FUNCTION_BLOCK FBRealtimeSupport
///SDOC/////////////////////////////////////////////////////////////////////////
//
//  FBRealtimeSupport.TcPOU      - Function Block - Real-time diagnostic data with analog data - AVT PLC 
//						Version 1
//  Author:         Mark Colvin                         Date: Sept 5, 2018
//
//	Beckhoff TC3 Structured Text for CX8190 PLC
//
//	includes features:
//		10 inker enables
///////////////////////////////////////////////////////////////////////SDOCEND//
VAR_INPUT
END_VAR
VAR_OUTPUT
END_VAR
VAR
	// === LOCAL DATA === NOT saved over power cycles
	Index		:WORD;	//temp fountain index 
	wCycleCount	:WORD;	//cycle count for ON time for inker/water adjustments
	nActualScaled: INT;
	iActual: INT;
	w_output_incr	:INT;
END_VAR
VAR CONSTANT
	FTN1		:WORD:= 0;	//constants for fountain indexes fro IO arrays in TBs
	FTN2		:WORD:= 1;
	FTN3		:WORD:= 2;
	FTN4		:WORD:= 3;
	FTN5		:WORD:= 4;
	FTN6		:WORD:= 5;
	FTN7		:WORD:= 6;
	FTN8		:WORD:= 7;
	FTN9		:WORD:= 8;
	FTN10	:WORD:= 9;
	wMotorTimeOn :WORD:=500;  //wMotorTimeOn, how long the output is ON for ONE motor adjustment(+ or -), 1000 = 1second
END_VAR


	 CASE GVL.mb_Output_Registers[GVL.REALTIME_DATA_SELECTION] OF		//this is user selection of fountain control to inspect/modify
	 0:	//do nothing here
	 
	 // Inker analog inputs and outputs
	 1:	Index := FTN1;		//assign temp index
		CASE GVL.mb_Output_Registers[GVL.INKERHARDWARETYPE] OF
(* 		GVL.SWPWTR_TIME:
			//GVL.mb_Output_Registers[GVL.REALTIME_PLC_A2D] :=	0;	//nothing to read with FB circuit, just move motor
			IF GVL.mb_Output_Coils[GVL.REALTIME_ADVANCE] THEN		//move the motor forward
				IF TRUE THEN							//test the FB for limit - can't do this, pass through
					GVL.mb_Output_Coils[GVL.InkSweepRUN +(FTN1 * GVL.BOOLRUNTIMEGROUPSIZE)] := 	TRUE; //next RUN will force to console target
					GVL_IO.InkMotorFwd[FTN1] := TRUE;				// turn on the advance output
					GVL_IO.InkMotorRvs[FTN1] := FALSE;
					wCycleCount := wCycleCount + 1;
					IF wCycleCount > wMotorTimeOn THEN				//done with timer?
						GVL_IO.InkMotorFwd[FTN1] := FALSE;		//turn off outputs
						GVL_IO.InkMotorRvs[FTN1] := FALSE;
						GVL.mb_Output_Coils[GVL.REALTIME_ADVANCE] := FALSE; // reset the advance boolean
						wCycleCount := 0;					//reset the timer counter						
					END_IF
				END_IF
			END_IF
			IF GVL.mb_Output_Coils[GVL.REALTIME_RETARD] THEN
				IF TRUE THEN							//test the FB for limit - can't do this, pass through
					GVL.mb_Output_Coils[GVL.InkSweepRUN +(FTN1 * GVL.BOOLRUNTIMEGROUPSIZE)] := 	TRUE; //next RUN will force to console target
					GVL_IO.InkMotorFwd[FTN1] := FALSE;				// turn on the reverse output
					GVL_IO.InkMotorRvs[FTN1] := TRUE;
					wCycleCount := wCycleCount + 1;
					IF wCycleCount > wMotorTimeOn THEN				//done with timer?
						GVL_IO.InkMotorFwd[FTN1] := FALSE;		//turn off outputs
						GVL_IO.InkMotorRvs[FTN1] := FALSE;
						GVL.mb_Output_Coils[GVL.REALTIME_RETARD] := FALSE; // reset the reverse boolean
						wCycleCount := 0;					//reset the timer counter						
					END_IF
				END_IF
			END_IF
		GVL.SWPWTR_FB:
			GVL.mb_Output_Registers[GVL.REALTIME_PLC_A2D] :=	INT_TO_WORD(GVL_IO.InkInput[FTN1]);
			IF GVL.mb_Output_Coils[GVL.REALTIME_ADVANCE] THEN		//move the motor forward
				IF INT_TO_WORD(GVL_IO.InkInput[FTN1]) < 32000 THEN				//test the FB for limit - assumes 32767 is max of 10 VDC
					GVL.mb_Output_Coils[GVL.InkSweepRUN +(FTN1 * GVL.BOOLRUNTIMEGROUPSIZE)] := 	TRUE; //next RUN will force to console target
					GVL_IO.InkMotorFwd[FTN1] := TRUE;				// turn on the advance output
					GVL_IO.InkMotorRvs[FTN1] := FALSE;
					wCycleCount := wCycleCount + 1;
					IF wCycleCount > wMotorTimeOn THEN				//done with timer?
						GVL_IO.InkMotorFwd[FTN1] := FALSE;		//turn off outputs
						GVL_IO.InkMotorRvs[FTN1] := FALSE;
						GVL.mb_Output_Coils[GVL.REALTIME_ADVANCE] := FALSE; // reset the advance boolean
						wCycleCount := 0;					//reset the timer counter	
						//  curr % sweep   curr ticks - min tick allowed      max sweep %            max ticks allowed      min ticks allowed
						GVL.mb_Output_Registers[GVL.SWEEPTRIMONPRESS + (FTN10 * GVL.WORDRUNTIMEGROUPSIZE)]	:= (INT_TO_WORD(GVL_IO.InkInput[FTN1]) - GVL.w_InkInputIntMin[FTN10]) * 
								(GVL.mb_Output_Registers[GVL.MAXSWEEPTRIM]+1) / (GVL.w_InkInputIntMax[FTN10] - GVL.w_InkInputIntMin[FTN10]);
						//need the onpress setting pointed to the current % sweep of the positioner
					END_IF
				END_IF
			END_IF
			IF GVL.mb_Output_Coils[GVL.REALTIME_RETARD] THEN
				IF INT_TO_WORD(GVL_IO.InkInput[FTN1]) > 800 THEN				//test the FB for limit - assumes 32767 is max of 10 VDC
					GVL.mb_Output_Coils[GVL.InkSweepRUN +(FTN1 * GVL.BOOLRUNTIMEGROUPSIZE)] := 	TRUE; //next RUN will force to console target
					GVL_IO.InkMotorFwd[FTN1] := FALSE;				// turn on the reverse output
					GVL_IO.InkMotorRvs[FTN1] := TRUE;
					wCycleCount := wCycleCount + 1;
					IF wCycleCount > wMotorTimeOn THEN				//done with timer?
						GVL_IO.InkMotorFwd[FTN1] := FALSE;		//turn off outputs
						GVL_IO.InkMotorRvs[FTN1] := FALSE;
						GVL.mb_Output_Coils[GVL.REALTIME_RETARD] := FALSE; // reset the reverse boolean
						wCycleCount := 0;					//reset the timer counter						
						//  curr % sweep   curr ticks - min tick allowed      max sweep %            max ticks allowed      min ticks allowed
						GVL.mb_Output_Registers[GVL.SWEEPTRIMONPRESS + (FTN1 * GVL.WORDRUNTIMEGROUPSIZE)]	:= (INT_TO_WORD(GVL_IO.InkInput[FTN1]) - GVL.w_InkInputIntMin[FTN1]) * 
								(GVL.mb_Output_Registers[GVL.MAXSWEEPTRIM]+1) / (GVL.w_InkInputIntMax[FTN1] - GVL.w_InkInputIntMin[FTN1]);
						//need the onpress setting pointed to the current % sweep of the positioner
					END_IF
				END_IF
			END_IF
		GVL.SWPWTR_OUTPUT:
			GVL.mb_Output_Registers[GVL.REALTIME_PLC_A2D] :=	INT_TO_WORD(GVL_IO.InkSweepOut[FTN1]);
			IF( GVL.b_DINTInput) THEN									//how big should the adv / ret control increment be?
				w_output_incr :=  DINT_TO_INT(GVL.d_DINT10V / 100);
			ELSE
				w_output_incr := (GVL.i_INT10V / 100);
			END_IF
			IF GVL.mb_Output_Coils[GVL.REALTIME_ADVANCE] THEN
				IF (GVL_IO.InkSweepOut[FTN1]) < (w_output_incr *100) THEN
					GVL.mb_Output_Coils[GVL.InkSweepRUN +(FTN1 * GVL.BOOLRUNTIMEGROUPSIZE)] := 	TRUE; //next RUN will force to console target
					GVL_IO.InkSweepOut[FTN1] := (GVL_IO.InkSweepOut[FTN1]) + w_output_incr;
				END_IF
				GVL.mb_Output_Coils[GVL.REALTIME_ADVANCE] := FALSE;
			END_IF
			IF GVL.mb_Output_Coils[GVL.REALTIME_RETARD] THEN
				IF (GVL_IO.InkSweepOut[FTN1]) > w_output_incr THEN
					GVL.mb_Output_Coils[GVL.InkSweepRUN +(FTN1 * GVL.BOOLRUNTIMEGROUPSIZE)] := 	TRUE; //next RUN will force to console target
					GVL_IO.InkSweepOut[FTN1] := (GVL_IO.InkSweepOut[FTN1]) - w_output_incr;
				END_IF
				GVL.mb_Output_Coils[GVL.REALTIME_RETARD] := FALSE;
			END_IF			
 *)
		GVL.SWPWTR_BRIDGE:

		END_CASE
	 2:	Index := FTN2;		//assign temp index
		CASE GVL.mb_Output_Registers[GVL.INKERHARDWARETYPE] OF
(* 		GVL.SWPWTR_TIME:
			//GVL.mb_Output_Registers[GVL.REALTIME_PLC_A2D] :=	0;	//nothing to read with FB circuit, just move motor
			IF GVL.mb_Output_Coils[GVL.REALTIME_ADVANCE] THEN		//move the motor forward
				IF TRUE THEN							//test the FB for limit - can't do this, pass through
					GVL.mb_Output_Coils[GVL.InkSweepRUN +(FTN2 * GVL.BOOLRUNTIMEGROUPSIZE)] := 	TRUE; //next RUN will force to console target
					GVL_IO.InkMotorFwd[FTN2] := TRUE;				// turn on the advance output
					GVL_IO.InkMotorRvs[FTN2] := FALSE;
					wCycleCount := wCycleCount + 1;
					IF wCycleCount > wMotorTimeOn THEN				//done with timer?
						GVL_IO.InkMotorFwd[FTN2] := FALSE;		//turn off outputs
						GVL_IO.InkMotorRvs[FTN2] := FALSE;
						GVL.mb_Output_Coils[GVL.REALTIME_ADVANCE] := FALSE; // reset the advance boolean
						wCycleCount := 0;					//reset the timer counter						
					END_IF
				END_IF
			END_IF
			IF GVL.mb_Output_Coils[GVL.REALTIME_RETARD] THEN
				IF TRUE THEN							//test the FB for limit - can't do this, pass through
					GVL.mb_Output_Coils[GVL.InkSweepRUN +(FTN2 * GVL.BOOLRUNTIMEGROUPSIZE)] := 	TRUE; //next RUN will force to console target
					GVL_IO.InkMotorFwd[FTN2] := FALSE;				// turn on the reverse output
					GVL_IO.InkMotorRvs[FTN2] := TRUE;
					wCycleCount := wCycleCount + 1;
					IF wCycleCount > wMotorTimeOn THEN				//done with timer?
						GVL_IO.InkMotorFwd[FTN2] := FALSE;		//turn off outputs
						GVL_IO.InkMotorRvs[FTN2] := FALSE;
						GVL.mb_Output_Coils[GVL.REALTIME_RETARD] := FALSE; // reset the reverse boolean
						wCycleCount := 0;					//reset the timer counter						
					END_IF
				END_IF
			END_IF
		GVL.SWPWTR_FB:
			GVL.mb_Output_Registers[GVL.REALTIME_PLC_A2D] :=	INT_TO_WORD(GVL_IO.InkInput[FTN2]);
			IF GVL.mb_Output_Coils[GVL.REALTIME_ADVANCE] THEN		//move the motor forward
				IF INT_TO_WORD(GVL_IO.InkInput[FTN2]) < 32000 THEN				//test the FB for limit - assumes 32767 is max of 10 VDC
					GVL.mb_Output_Coils[GVL.InkSweepRUN +(FTN2 * GVL.BOOLRUNTIMEGROUPSIZE)] := 	TRUE; //next RUN will force to console target
					GVL_IO.InkMotorFwd[FTN2] := TRUE;				// turn on the advance output
					GVL_IO.InkMotorRvs[FTN2] := FALSE;
					wCycleCount := wCycleCount + 1;
					IF wCycleCount > wMotorTimeOn THEN				//done with timer?
						GVL_IO.InkMotorFwd[FTN2] := FALSE;		//turn off outputs
						GVL_IO.InkMotorRvs[FTN2] := FALSE;
						GVL.mb_Output_Coils[GVL.REALTIME_ADVANCE] := FALSE; // reset the advance boolean
						wCycleCount := 0;					//reset the timer counter	
						//  curr % sweep   curr ticks - min tick allowed      max sweep %            max ticks allowed      min ticks allowed
						GVL.mb_Output_Registers[GVL.SWEEPTRIMONPRESS + (FTN2 * GVL.WORDRUNTIMEGROUPSIZE)]	:= (INT_TO_WORD(GVL_IO.InkInput[FTN2]) - GVL.w_InkInputIntMin[FTN2]) * 
								(GVL.mb_Output_Registers[GVL.MAXSWEEPTRIM]+1) / (GVL.w_InkInputIntMax[FTN2] - GVL.w_InkInputIntMin[FTN2]);
						//need the onpress setting pointed to the current % sweep of the positioner
					END_IF
				END_IF
			END_IF
			IF GVL.mb_Output_Coils[GVL.REALTIME_RETARD] THEN
				IF INT_TO_WORD(GVL_IO.InkInput[FTN2]) > 800 THEN				//test the FB for limit - assumes 32767 is max of 10 VDC
					GVL.mb_Output_Coils[GVL.InkSweepRUN +(FTN2 * GVL.BOOLRUNTIMEGROUPSIZE)] := 	TRUE; //next RUN will force to console target
					GVL_IO.InkMotorFwd[FTN2] := FALSE;				// turn on the reverse output
					GVL_IO.InkMotorRvs[FTN2] := TRUE;
					wCycleCount := wCycleCount + 1;
					IF wCycleCount > wMotorTimeOn THEN				//done with timer?
						GVL_IO.InkMotorFwd[FTN2] := FALSE;		//turn off outputs
						GVL_IO.InkMotorRvs[FTN2] := FALSE;
						GVL.mb_Output_Coils[GVL.REALTIME_RETARD] := FALSE; // reset the reverse boolean
						wCycleCount := 0;					//reset the timer counter						
						//  curr % sweep   curr ticks - min tick allowed      max sweep %            max ticks allowed      min ticks allowed
						GVL.mb_Output_Registers[GVL.SWEEPTRIMONPRESS + (FTN2 * GVL.WORDRUNTIMEGROUPSIZE)]	:= (INT_TO_WORD(GVL_IO.InkInput[FTN2]) - GVL.w_InkInputIntMin[FTN2]) * 
								(GVL.mb_Output_Registers[GVL.MAXSWEEPTRIM]+1) / (GVL.w_InkInputIntMax[FTN2] - GVL.w_InkInputIntMin[FTN2]);
						//need the onpress setting pointed to the current % sweep of the positioner
					END_IF
				END_IF
			END_IF
		GVL.SWPWTR_OUTPUT:
			GVL.mb_Output_Registers[GVL.REALTIME_PLC_A2D] :=	INT_TO_WORD(GVL_IO.InkSweepOut[FTN2]);
			IF( GVL.b_DINTInput) THEN									//how big should the adv / ret control increment be?
				w_output_incr :=  DINT_TO_INT(GVL.d_DINT10V / 100);
			ELSE
				w_output_incr := (GVL.i_INT10V / 100);
			END_IF
			IF GVL.mb_Output_Coils[GVL.REALTIME_ADVANCE] THEN
				IF GVL_IO.InkSweepOut[FTN2] < (w_output_incr *100) THEN
					GVL.mb_Output_Coils[GVL.InkSweepRUN +(FTN2 * GVL.BOOLRUNTIMEGROUPSIZE)] := 	TRUE; //next RUN will force to console target
					GVL_IO.InkSweepOut[FTN2] := GVL_IO.InkSweepOut[FTN2] + w_output_incr;
				END_IF
				GVL.mb_Output_Coils[GVL.REALTIME_ADVANCE] := FALSE;
			END_IF
			IF GVL.mb_Output_Coils[GVL.REALTIME_RETARD] THEN
				IF GVL_IO.InkSweepOut[FTN2] > w_output_incr THEN
					GVL.mb_Output_Coils[GVL.InkSweepRUN +(FTN2 * GVL.BOOLRUNTIMEGROUPSIZE)] := 	TRUE; //next RUN will force to console target
					GVL_IO.InkSweepOut[FTN2] := GVL_IO.InkSweepOut[FTN2] - w_output_incr;
				END_IF
				GVL.mb_Output_Coils[GVL.REALTIME_RETARD] := FALSE;
			END_IF			
 *)
		GVL.SWPWTR_BRIDGE:
		END_CASE
	 3:	Index := FTN3;		//assign temp index
		CASE GVL.mb_Output_Registers[GVL.INKERHARDWARETYPE] OF
(* 		GVL.SWPWTR_TIME:
			//GVL.mb_Output_Registers[GVL.REALTIME_PLC_A2D] :=	0;	//nothing to read with FB circuit, just move motor
			IF GVL.mb_Output_Coils[GVL.REALTIME_ADVANCE] THEN		//move the motor forward
				IF TRUE THEN							//test the FB for limit - can't do this, pass through
					GVL.mb_Output_Coils[GVL.InkSweepRUN +(FTN3 * GVL.BOOLRUNTIMEGROUPSIZE)] := 	TRUE; //next RUN will force to console target
					GVL_IO.InkMotorFwd[FTN3] := TRUE;				// turn on the advance output
					GVL_IO.InkMotorRvs[FTN3] := FALSE;
					wCycleCount := wCycleCount + 1;
					IF wCycleCount > wMotorTimeOn THEN				//done with timer?
						GVL_IO.InkMotorFwd[FTN3] := FALSE;		//turn off outputs
						GVL_IO.InkMotorRvs[FTN3] := FALSE;
						GVL.mb_Output_Coils[GVL.REALTIME_ADVANCE] := FALSE; // reset the advance boolean
						wCycleCount := 0;					//reset the timer counter						
					END_IF
				END_IF
			END_IF
			IF GVL.mb_Output_Coils[GVL.REALTIME_RETARD] THEN
				IF TRUE THEN							//test the FB for limit - can't do this, pass through
					GVL.mb_Output_Coils[GVL.InkSweepRUN +(FTN3 * GVL.BOOLRUNTIMEGROUPSIZE)] := 	TRUE; //next RUN will force to console target
					GVL_IO.InkMotorFwd[FTN3] := FALSE;				// turn on the reverse output
					GVL_IO.InkMotorRvs[FTN3] := TRUE;
					wCycleCount := wCycleCount + 1;
					IF wCycleCount > wMotorTimeOn THEN				//done with timer?
						GVL_IO.InkMotorFwd[FTN3] := FALSE;		//turn off outputs
						GVL_IO.InkMotorRvs[FTN3] := FALSE;
						GVL.mb_Output_Coils[GVL.REALTIME_RETARD] := FALSE; // reset the reverse boolean
						wCycleCount := 0;					//reset the timer counter						
					END_IF
				END_IF
			END_IF
		GVL.SWPWTR_FB:
			GVL.mb_Output_Registers[GVL.REALTIME_PLC_A2D] :=	INT_TO_WORD(GVL_IO.InkInput[FTN3]);
			IF GVL.mb_Output_Coils[GVL.REALTIME_ADVANCE] THEN		//move the motor forward
				IF INT_TO_WORD(GVL_IO.InkInput[FTN3]) < 32000 THEN				//test the FB for limit - assumes 32767 is max of 10 VDC
					GVL.mb_Output_Coils[GVL.InkSweepRUN +(FTN3 * GVL.BOOLRUNTIMEGROUPSIZE)] := 	TRUE; //next RUN will force to console target
					GVL_IO.InkMotorFwd[FTN3] := TRUE;				// turn on the advance output
					GVL_IO.InkMotorRvs[FTN3] := FALSE;
					wCycleCount := wCycleCount + 1;
					IF wCycleCount > wMotorTimeOn THEN				//done with timer?
						GVL_IO.InkMotorFwd[FTN3] := FALSE;		//turn off outputs
						GVL_IO.InkMotorRvs[FTN3] := FALSE;
						GVL.mb_Output_Coils[GVL.REALTIME_ADVANCE] := FALSE; // reset the advance boolean
						wCycleCount := 0;					//reset the timer counter	
						//  curr % sweep   curr ticks - min tick allowed      max sweep %            max ticks allowed      min ticks allowed
						GVL.mb_Output_Registers[GVL.SWEEPTRIMONPRESS + (FTN3 * GVL.WORDRUNTIMEGROUPSIZE)]	:= (INT_TO_WORD(GVL_IO.InkInput[FTN3]) - GVL.w_InkInputIntMin[FTN3]) * 
								(GVL.mb_Output_Registers[GVL.MAXSWEEPTRIM]+1) / (GVL.w_InkInputIntMax[FTN3] - GVL.w_InkInputIntMin[FTN3]);
						//need the onpress setting pointed to the current % sweep of the positioner
					END_IF
				END_IF
			END_IF
			IF GVL.mb_Output_Coils[GVL.REALTIME_RETARD] THEN
				IF INT_TO_WORD(GVL_IO.InkInput[FTN3]) > 800 THEN				//test the FB for limit - assumes 32767 is max of 10 VDC
					GVL.mb_Output_Coils[GVL.InkSweepRUN +(FTN3 * GVL.BOOLRUNTIMEGROUPSIZE)] := 	TRUE; //next RUN will force to console target
					GVL_IO.InkMotorFwd[FTN3] := FALSE;				// turn on the reverse output
					GVL_IO.InkMotorRvs[FTN3] := TRUE;
					wCycleCount := wCycleCount + 1;
					IF wCycleCount > wMotorTimeOn THEN				//done with timer?
						GVL_IO.InkMotorFwd[FTN3] := FALSE;		//turn off outputs
						GVL_IO.InkMotorRvs[FTN3] := FALSE;
						GVL.mb_Output_Coils[GVL.REALTIME_RETARD] := FALSE; // reset the reverse boolean
						wCycleCount := 0;					//reset the timer counter						
						//  curr % sweep   curr ticks - min tick allowed      max sweep %            max ticks allowed      min ticks allowed
						GVL.mb_Output_Registers[GVL.SWEEPTRIMONPRESS + (FTN3 * GVL.WORDRUNTIMEGROUPSIZE)]	:= (INT_TO_WORD(GVL_IO.InkInput[FTN3]) - GVL.w_InkInputIntMin[FTN3]) * 
								(GVL.mb_Output_Registers[GVL.MAXSWEEPTRIM]+1) / (GVL.w_InkInputIntMax[FTN3] - GVL.w_InkInputIntMin[FTN3]);
						//need the onpress setting pointed to the current % sweep of the positioner
					END_IF
				END_IF
			END_IF
		GVL.SWPWTR_OUTPUT:
			GVL.mb_Output_Registers[GVL.REALTIME_PLC_A2D] :=	INT_TO_WORD(GVL_IO.InkSweepOut[FTN3]);
			IF( GVL.b_DINTInput) THEN									//how big should the adv / ret control increment be?
				w_output_incr :=  DINT_TO_INT(GVL.d_DINT10V / 100);
			ELSE
				w_output_incr := (GVL.i_INT10V / 100);
			END_IF
			IF GVL.mb_Output_Coils[GVL.REALTIME_ADVANCE] THEN
				IF GVL_IO.InkSweepOut[FTN3] < (w_output_incr *100) THEN
					GVL.mb_Output_Coils[GVL.InkSweepRUN +(FTN3 * GVL.BOOLRUNTIMEGROUPSIZE)] := 	TRUE; //next RUN will force to console target
					GVL_IO.InkSweepOut[FTN3] := GVL_IO.InkSweepOut[FTN3] + w_output_incr;
				END_IF
				GVL.mb_Output_Coils[GVL.REALTIME_ADVANCE] := FALSE;
			END_IF
			IF GVL.mb_Output_Coils[GVL.REALTIME_RETARD] THEN
				IF GVL_IO.InkSweepOut[FTN3] > w_output_incr THEN
					GVL.mb_Output_Coils[GVL.InkSweepRUN +(FTN3 * GVL.BOOLRUNTIMEGROUPSIZE)] := 	TRUE; //next RUN will force to console target
					GVL_IO.InkSweepOut[FTN3] := GVL_IO.InkSweepOut[FTN3] - w_output_incr;
				END_IF
				GVL.mb_Output_Coils[GVL.REALTIME_RETARD] := FALSE;
			END_IF			
 *)		
		GVL.SWPWTR_BRIDGE:
		END_CASE
	 4:	Index := FTN4;		//assign temp index
		CASE GVL.mb_Output_Registers[GVL.INKERHARDWARETYPE] OF
(* 		GVL.SWPWTR_TIME:
			//GVL.mb_Output_Registers[GVL.REALTIME_PLC_A2D] :=	0;	//nothing to read with FB circuit, just move motor
			IF GVL.mb_Output_Coils[GVL.REALTIME_ADVANCE] THEN		//move the motor forward
				IF TRUE THEN							//test the FB for limit - can't do this, pass through
					GVL.mb_Output_Coils[GVL.InkSweepRUN +(FTN4 * GVL.BOOLRUNTIMEGROUPSIZE)] := 	TRUE; //next RUN will force to console target
					GVL_IO.InkMotorFwd[FTN4] := TRUE;				// turn on the advance output
					GVL_IO.InkMotorRvs[FTN4] := FALSE;
					wCycleCount := wCycleCount + 1;
					IF wCycleCount > wMotorTimeOn THEN				//done with timer?
						GVL_IO.InkMotorFwd[FTN4] := FALSE;		//turn off outputs
						GVL_IO.InkMotorRvs[FTN4] := FALSE;
						GVL.mb_Output_Coils[GVL.REALTIME_ADVANCE] := FALSE; // reset the advance boolean
						wCycleCount := 0;					//reset the timer counter						
					END_IF
				END_IF
			END_IF
			IF GVL.mb_Output_Coils[GVL.REALTIME_RETARD] THEN
				IF TRUE THEN							//test the FB for limit - can't do this, pass through
					GVL.mb_Output_Coils[GVL.InkSweepRUN +(FTN4 * GVL.BOOLRUNTIMEGROUPSIZE)] := 	TRUE; //next RUN will force to console target
					GVL_IO.InkMotorFwd[FTN4] := FALSE;				// turn on the reverse output
					GVL_IO.InkMotorRvs[FTN4] := TRUE;
					wCycleCount := wCycleCount + 1;
					IF wCycleCount > wMotorTimeOn THEN				//done with timer?
						GVL_IO.InkMotorFwd[FTN4] := FALSE;		//turn off outputs
						GVL_IO.InkMotorRvs[FTN4] := FALSE;
						GVL.mb_Output_Coils[GVL.REALTIME_RETARD] := FALSE; // reset the reverse boolean
						wCycleCount := 0;					//reset the timer counter						
					END_IF
				END_IF
			END_IF
		GVL.SWPWTR_FB:
			GVL.mb_Output_Registers[GVL.REALTIME_PLC_A2D] :=	INT_TO_WORD(GVL_IO.InkInput[FTN4]);
			IF GVL.mb_Output_Coils[GVL.REALTIME_ADVANCE] THEN		//move the motor forward
				IF INT_TO_WORD(GVL_IO.InkInput[FTN4]) < 32000 THEN				//test the FB for limit - assumes 32767 is max of 10 VDC
					GVL.mb_Output_Coils[GVL.InkSweepRUN +(FTN4 * GVL.BOOLRUNTIMEGROUPSIZE)] := 	TRUE; //next RUN will force to console target
					GVL_IO.InkMotorFwd[FTN4] := TRUE;				// turn on the advance output
					GVL_IO.InkMotorRvs[FTN4] := FALSE;
					wCycleCount := wCycleCount + 1;
					IF wCycleCount > wMotorTimeOn THEN				//done with timer?
						GVL_IO.InkMotorFwd[FTN4] := FALSE;		//turn off outputs
						GVL_IO.InkMotorRvs[FTN4] := FALSE;
						GVL.mb_Output_Coils[GVL.REALTIME_ADVANCE] := FALSE; // reset the advance boolean
						wCycleCount := 0;					//reset the timer counter	
						//  curr % sweep   curr ticks - min tick allowed      max sweep %            max ticks allowed      min ticks allowed
						GVL.mb_Output_Registers[GVL.SWEEPTRIMONPRESS + (FTN4 * GVL.WORDRUNTIMEGROUPSIZE)]	:= (INT_TO_WORD(GVL_IO.InkInput[FTN4]) - GVL.w_InkInputIntMin[FTN4]) * 
								(GVL.mb_Output_Registers[GVL.MAXSWEEPTRIM]+1) / (GVL.w_InkInputIntMax[FTN4] - GVL.w_InkInputIntMin[FTN4]);
						//need the onpress setting pointed to the current % sweep of the positioner
					END_IF
				END_IF
			END_IF
			IF GVL.mb_Output_Coils[GVL.REALTIME_RETARD] THEN
				IF INT_TO_WORD(GVL_IO.InkInput[FTN4]) > 800 THEN				//test the FB for limit - assumes 32767 is max of 10 VDC
					GVL.mb_Output_Coils[GVL.InkSweepRUN +(FTN4 * GVL.BOOLRUNTIMEGROUPSIZE)] := 	TRUE; //next RUN will force to console target
					GVL_IO.InkMotorFwd[FTN4] := FALSE;				// turn on the reverse output
					GVL_IO.InkMotorRvs[FTN4] := TRUE;
					wCycleCount := wCycleCount + 1;
					IF wCycleCount > wMotorTimeOn THEN				//done with timer?
						GVL_IO.InkMotorFwd[FTN4] := FALSE;		//turn off outputs
						GVL_IO.InkMotorRvs[FTN4] := FALSE;
						GVL.mb_Output_Coils[GVL.REALTIME_RETARD] := FALSE; // reset the reverse boolean
						wCycleCount := 0;					//reset the timer counter						
						//  curr % sweep   curr ticks - min tick allowed      max sweep %            max ticks allowed      min ticks allowed
						GVL.mb_Output_Registers[GVL.SWEEPTRIMONPRESS + (FTN4 * GVL.WORDRUNTIMEGROUPSIZE)]	:= (INT_TO_WORD(GVL_IO.InkInput[FTN4]) - GVL.w_InkInputIntMin[FTN4]) * 
								(GVL.mb_Output_Registers[GVL.MAXSWEEPTRIM]+1) / (GVL.w_InkInputIntMax[FTN4] - GVL.w_InkInputIntMin[FTN4]);
						//need the onpress setting pointed to the current % sweep of the positioner
					END_IF
				END_IF
			END_IF
		GVL.SWPWTR_OUTPUT:
			GVL.mb_Output_Registers[GVL.REALTIME_PLC_A2D] :=	INT_TO_WORD(GVL_IO.InkSweepOut[FTN4]);
			IF( GVL.b_DINTInput) THEN									//how big should the adv / ret control increment be?
				w_output_incr :=  DINT_TO_INT(GVL.d_DINT10V / 100);
			ELSE
				w_output_incr := (GVL.i_INT10V / 100);
			END_IF
			IF GVL.mb_Output_Coils[GVL.REALTIME_ADVANCE] THEN
				IF GVL_IO.InkSweepOut[FTN4] < (w_output_incr *100) THEN
					GVL.mb_Output_Coils[GVL.InkSweepRUN +(FTN4 * GVL.BOOLRUNTIMEGROUPSIZE)] := 	TRUE; //next RUN will force to console target
					GVL_IO.InkSweepOut[FTN4] := GVL_IO.InkSweepOut[FTN4] + w_output_incr;
				END_IF
				GVL.mb_Output_Coils[GVL.REALTIME_ADVANCE] := FALSE;
			END_IF
			IF GVL.mb_Output_Coils[GVL.REALTIME_RETARD] THEN
				IF GVL_IO.InkSweepOut[FTN4] > w_output_incr THEN
					GVL.mb_Output_Coils[GVL.InkSweepRUN +(FTN4 * GVL.BOOLRUNTIMEGROUPSIZE)] := 	TRUE; //next RUN will force to console target
					GVL_IO.InkSweepOut[FTN4] := GVL_IO.InkSweepOut[FTN4] - w_output_incr;
				END_IF
				GVL.mb_Output_Coils[GVL.REALTIME_RETARD] := FALSE;
			END_IF			
 *)
		GVL.SWPWTR_BRIDGE:
		END_CASE
	 5:	Index := FTN5;		//assign temp index
		CASE GVL.mb_Output_Registers[GVL.INKERHARDWARETYPE] OF
(* 		GVL.SWPWTR_TIME:
			//GVL.mb_Output_Registers[GVL.REALTIME_PLC_A2D] :=	0;	//nothing to read with FB circuit, just move motor
			IF GVL.mb_Output_Coils[GVL.REALTIME_ADVANCE] THEN		//move the motor forward
				IF TRUE THEN							//test the FB for limit - can't do this, pass through
					GVL.mb_Output_Coils[GVL.InkSweepRUN +(FTN5 * GVL.BOOLRUNTIMEGROUPSIZE)] := 	TRUE; //next RUN will force to console target
					GVL_IO.InkMotorFwd[FTN5] := TRUE;				// turn on the advance output
					GVL_IO.InkMotorRvs[FTN5] := FALSE;
					wCycleCount := wCycleCount + 1;
					IF wCycleCount > wMotorTimeOn THEN				//done with timer?
						GVL_IO.InkMotorFwd[FTN5] := FALSE;		//turn off outputs
						GVL_IO.InkMotorRvs[FTN5] := FALSE;
						GVL.mb_Output_Coils[GVL.REALTIME_ADVANCE] := FALSE; // reset the advance boolean
						wCycleCount := 0;					//reset the timer counter						
					END_IF
				END_IF
			END_IF
			IF GVL.mb_Output_Coils[GVL.REALTIME_RETARD] THEN
				IF TRUE THEN							//test the FB for limit - can't do this, pass through
					GVL.mb_Output_Coils[GVL.InkSweepRUN +(FTN5 * GVL.BOOLRUNTIMEGROUPSIZE)] := 	TRUE; //next RUN will force to console target
					GVL_IO.InkMotorFwd[FTN5] := FALSE;				// turn on the reverse output
					GVL_IO.InkMotorRvs[FTN5] := TRUE;
					wCycleCount := wCycleCount + 1;
					IF wCycleCount > wMotorTimeOn THEN				//done with timer?
						GVL_IO.InkMotorFwd[FTN5] := FALSE;		//turn off outputs
						GVL_IO.InkMotorRvs[FTN5] := FALSE;
						GVL.mb_Output_Coils[GVL.REALTIME_RETARD] := FALSE; // reset the reverse boolean
						wCycleCount := 0;					//reset the timer counter						
					END_IF
				END_IF
			END_IF
		GVL.SWPWTR_FB:
			GVL.mb_Output_Registers[GVL.REALTIME_PLC_A2D] :=	INT_TO_WORD(GVL_IO.InkInput[FTN5]);
			IF GVL.mb_Output_Coils[GVL.REALTIME_ADVANCE] THEN		//move the motor forward
				IF INT_TO_WORD(GVL_IO.InkInput[FTN5]) < 32000 THEN				//test the FB for limit - assumes 32767 is max of 10 VDC
					GVL.mb_Output_Coils[GVL.InkSweepRUN +(FTN5 * GVL.BOOLRUNTIMEGROUPSIZE)] := 	TRUE; //next RUN will force to console target
					GVL_IO.InkMotorFwd[FTN5] := TRUE;				// turn on the advance output
					GVL_IO.InkMotorRvs[FTN5] := FALSE;
					wCycleCount := wCycleCount + 1;
					IF wCycleCount > wMotorTimeOn THEN				//done with timer?
						GVL_IO.InkMotorFwd[FTN5] := FALSE;		//turn off outputs
						GVL_IO.InkMotorRvs[FTN5] := FALSE;
						GVL.mb_Output_Coils[GVL.REALTIME_ADVANCE] := FALSE; // reset the advance boolean
						wCycleCount := 0;					//reset the timer counter	
						//  curr % sweep   curr ticks - min tick allowed      max sweep %            max ticks allowed      min ticks allowed
						GVL.mb_Output_Registers[GVL.SWEEPTRIMONPRESS + (FTN5 * GVL.WORDRUNTIMEGROUPSIZE)]	:= (INT_TO_WORD(GVL_IO.InkInput[FTN5]) - GVL.w_InkInputIntMin[FTN5]) * 
								(GVL.mb_Output_Registers[GVL.MAXSWEEPTRIM]+1) / (GVL.w_InkInputIntMax[FTN5] - GVL.w_InkInputIntMin[FTN5]);
						//need the onpress setting pointed to the current % sweep of the positioner
					END_IF
				END_IF
			END_IF
			IF GVL.mb_Output_Coils[GVL.REALTIME_RETARD] THEN
				IF INT_TO_WORD(GVL_IO.InkInput[FTN5]) > 800 THEN				//test the FB for limit - assumes 32767 is max of 10 VDC
					GVL.mb_Output_Coils[GVL.InkSweepRUN +(FTN5 * GVL.BOOLRUNTIMEGROUPSIZE)] := 	TRUE; //next RUN will force to console target
					GVL_IO.InkMotorFwd[FTN5] := FALSE;				// turn on the reverse output
					GVL_IO.InkMotorRvs[FTN5] := TRUE;
					wCycleCount := wCycleCount + 1;
					IF wCycleCount > wMotorTimeOn THEN				//done with timer?
						GVL_IO.InkMotorFwd[FTN5] := FALSE;		//turn off outputs
						GVL_IO.InkMotorRvs[FTN5] := FALSE;
						GVL.mb_Output_Coils[GVL.REALTIME_RETARD] := FALSE; // reset the reverse boolean
						wCycleCount := 0;					//reset the timer counter						
						//  curr % sweep   curr ticks - min tick allowed      max sweep %            max ticks allowed      min ticks allowed
						GVL.mb_Output_Registers[GVL.SWEEPTRIMONPRESS + (FTN5 * GVL.WORDRUNTIMEGROUPSIZE)]	:= (INT_TO_WORD(GVL_IO.InkInput[FTN5]) - GVL.w_InkInputIntMin[FTN5]) * 
								(GVL.mb_Output_Registers[GVL.MAXSWEEPTRIM]+1) / (GVL.w_InkInputIntMax[FTN5] - GVL.w_InkInputIntMin[FTN5]);
						//need the onpress setting pointed to the current % sweep of the positioner
					END_IF
				END_IF
			END_IF
		GVL.SWPWTR_OUTPUT:
			GVL.mb_Output_Registers[GVL.REALTIME_PLC_A2D] :=	INT_TO_WORD(GVL_IO.InkSweepOut[FTN5]);
			IF( GVL.b_DINTInput) THEN									//how big should the adv / ret control increment be?
				w_output_incr :=  DINT_TO_INT(GVL.d_DINT10V / 100);
			ELSE
				w_output_incr := (GVL.i_INT10V / 100);
			END_IF
			IF GVL.mb_Output_Coils[GVL.REALTIME_ADVANCE] THEN
				IF GVL_IO.InkSweepOut[FTN5] < (w_output_incr *100) THEN
					GVL.mb_Output_Coils[GVL.InkSweepRUN +(FTN5 * GVL.BOOLRUNTIMEGROUPSIZE)] := 	TRUE; //next RUN will force to console target
					GVL_IO.InkSweepOut[FTN5] := GVL_IO.InkSweepOut[FTN5] + w_output_incr;
				END_IF
				GVL.mb_Output_Coils[GVL.REALTIME_ADVANCE] := FALSE;
			END_IF
			IF GVL.mb_Output_Coils[GVL.REALTIME_RETARD] THEN
				IF GVL_IO.InkSweepOut[FTN5] > w_output_incr THEN
					GVL.mb_Output_Coils[GVL.InkSweepRUN +(FTN5 * GVL.BOOLRUNTIMEGROUPSIZE)] := 	TRUE; //next RUN will force to console target
					GVL_IO.InkSweepOut[FTN5] := GVL_IO.InkSweepOut[FTN5] - w_output_incr;
				END_IF
				GVL.mb_Output_Coils[GVL.REALTIME_RETARD] := FALSE;
			END_IF			
 *)
		GVL.SWPWTR_BRIDGE:
		END_CASE
	 6:	Index := FTN6;		//assign temp index
		CASE GVL.mb_Output_Registers[GVL.INKERHARDWARETYPE] OF
(* 		GVL.SWPWTR_TIME:
			//GVL.mb_Output_Registers[GVL.REALTIME_PLC_A2D] :=	0;	//nothing to read with FB circuit, just move motor
			IF GVL.mb_Output_Coils[GVL.REALTIME_ADVANCE] THEN		//move the motor forward
				IF TRUE THEN							//test the FB for limit - can't do this, pass through
					GVL.mb_Output_Coils[GVL.InkSweepRUN +(FTN6 * GVL.BOOLRUNTIMEGROUPSIZE)] := 	TRUE; //next RUN will force to console target
					GVL_IO.InkMotorFwd[FTN6] := TRUE;				// turn on the advance output
					GVL_IO.InkMotorRvs[FTN6] := FALSE;
					wCycleCount := wCycleCount + 1;
					IF wCycleCount > wMotorTimeOn THEN				//done with timer?
						GVL_IO.InkMotorFwd[FTN6] := FALSE;		//turn off outputs
						GVL_IO.InkMotorRvs[FTN6] := FALSE;
						GVL.mb_Output_Coils[GVL.REALTIME_ADVANCE] := FALSE; // reset the advance boolean
						wCycleCount := 0;					//reset the timer counter						
					END_IF
				END_IF
			END_IF
			IF GVL.mb_Output_Coils[GVL.REALTIME_RETARD] THEN
				IF TRUE THEN							//test the FB for limit - can't do this, pass through
					GVL.mb_Output_Coils[GVL.InkSweepRUN +(FTN6 * GVL.BOOLRUNTIMEGROUPSIZE)] := 	TRUE; //next RUN will force to console target
					GVL_IO.InkMotorFwd[FTN6] := FALSE;				// turn on the reverse output
					GVL_IO.InkMotorRvs[FTN6] := TRUE;
					wCycleCount := wCycleCount + 1;
					IF wCycleCount > wMotorTimeOn THEN				//done with timer?
						GVL_IO.InkMotorFwd[FTN6] := FALSE;		//turn off outputs
						GVL_IO.InkMotorRvs[FTN6] := FALSE;
						GVL.mb_Output_Coils[GVL.REALTIME_RETARD] := FALSE; // reset the reverse boolean
						wCycleCount := 0;					//reset the timer counter						
					END_IF
				END_IF
			END_IF
		GVL.SWPWTR_FB:
			GVL.mb_Output_Registers[GVL.REALTIME_PLC_A2D] :=	INT_TO_WORD(GVL_IO.InkInput[FTN6]);
			IF GVL.mb_Output_Coils[GVL.REALTIME_ADVANCE] THEN		//move the motor forward
				IF INT_TO_WORD(GVL_IO.InkInput[FTN6]) < 32000 THEN				//test the FB for limit - assumes 32767 is max of 10 VDC
					GVL.mb_Output_Coils[GVL.InkSweepRUN +(FTN6 * GVL.BOOLRUNTIMEGROUPSIZE)] := 	TRUE; //next RUN will force to console target
					GVL_IO.InkMotorFwd[FTN6] := TRUE;				// turn on the advance output
					GVL_IO.InkMotorRvs[FTN6] := FALSE;
					wCycleCount := wCycleCount + 1;
					IF wCycleCount > wMotorTimeOn THEN				//done with timer?
						GVL_IO.InkMotorFwd[FTN6] := FALSE;		//turn off outputs
						GVL_IO.InkMotorRvs[FTN6] := FALSE;
						GVL.mb_Output_Coils[GVL.REALTIME_ADVANCE] := FALSE; // reset the advance boolean
						wCycleCount := 0;					//reset the timer counter	
						//  curr % sweep   curr ticks - min tick allowed      max sweep %            max ticks allowed      min ticks allowed
						GVL.mb_Output_Registers[GVL.SWEEPTRIMONPRESS + (FTN6 * GVL.WORDRUNTIMEGROUPSIZE)]	:= (INT_TO_WORD(GVL_IO.InkInput[FTN6]) - GVL.w_InkInputIntMin[FTN6]) * 
								(GVL.mb_Output_Registers[GVL.MAXSWEEPTRIM]+1) / (GVL.w_InkInputIntMax[FTN6] - GVL.w_InkInputIntMin[FTN6]);
						//need the onpress setting pointed to the current % sweep of the positioner
					END_IF
				END_IF
			END_IF
			IF GVL.mb_Output_Coils[GVL.REALTIME_RETARD] THEN
				IF INT_TO_WORD(GVL_IO.InkInput[FTN6]) > 800 THEN				//test the FB for limit - assumes 32767 is max of 10 VDC
					GVL.mb_Output_Coils[GVL.InkSweepRUN +(FTN6 * GVL.BOOLRUNTIMEGROUPSIZE)] := 	TRUE; //next RUN will force to console target
					GVL_IO.InkMotorFwd[FTN6] := FALSE;				// turn on the reverse output
					GVL_IO.InkMotorRvs[FTN6] := TRUE;
					wCycleCount := wCycleCount + 1;
					IF wCycleCount > wMotorTimeOn THEN				//done with timer?
						GVL_IO.InkMotorFwd[FTN6] := FALSE;		//turn off outputs
						GVL_IO.InkMotorRvs[FTN6] := FALSE;
						GVL.mb_Output_Coils[GVL.REALTIME_RETARD] := FALSE; // reset the reverse boolean
						wCycleCount := 0;					//reset the timer counter						
						//  curr % sweep   curr ticks - min tick allowed      max sweep %            max ticks allowed      min ticks allowed
						GVL.mb_Output_Registers[GVL.SWEEPTRIMONPRESS + (FTN6 * GVL.WORDRUNTIMEGROUPSIZE)]	:= (INT_TO_WORD(GVL_IO.InkInput[FTN6]) - GVL.w_InkInputIntMin[FTN6]) * 
								(GVL.mb_Output_Registers[GVL.MAXSWEEPTRIM]+1) / (GVL.w_InkInputIntMax[FTN6] - GVL.w_InkInputIntMin[FTN6]);
						//need the onpress setting pointed to the current % sweep of the positioner
					END_IF
				END_IF
			END_IF
		GVL.SWPWTR_OUTPUT:
			GVL.mb_Output_Registers[GVL.REALTIME_PLC_A2D] :=	INT_TO_WORD(GVL_IO.InkSweepOut[FTN6]);
			IF( GVL.b_DINTInput) THEN									//how big should the adv / ret control increment be?
				w_output_incr :=  DINT_TO_INT(GVL.d_DINT10V / 100);
			ELSE
				w_output_incr := (GVL.i_INT10V / 100);
			END_IF
			IF GVL.mb_Output_Coils[GVL.REALTIME_ADVANCE] THEN
				IF GVL_IO.InkSweepOut[FTN6] < (w_output_incr *100) THEN
					GVL.mb_Output_Coils[GVL.InkSweepRUN +(FTN6 * GVL.BOOLRUNTIMEGROUPSIZE)] := 	TRUE; //next RUN will force to console target
					GVL_IO.InkSweepOut[FTN6] := GVL_IO.InkSweepOut[FTN6] + w_output_incr;
				END_IF
				GVL.mb_Output_Coils[GVL.REALTIME_ADVANCE] := FALSE;
			END_IF
			IF GVL.mb_Output_Coils[GVL.REALTIME_RETARD] THEN
				IF GVL_IO.InkSweepOut[FTN6] > w_output_incr THEN
					GVL.mb_Output_Coils[GVL.InkSweepRUN +(FTN6 * GVL.BOOLRUNTIMEGROUPSIZE)] := 	TRUE; //next RUN will force to console target
					GVL_IO.InkSweepOut[FTN6] := GVL_IO.InkSweepOut[FTN6] - w_output_incr;
				END_IF
				GVL.mb_Output_Coils[GVL.REALTIME_RETARD] := FALSE;
			END_IF			
 *)
		GVL.SWPWTR_BRIDGE:
		END_CASE
	 7:	Index := FTN7;		//assign temp index
		CASE GVL.mb_Output_Registers[GVL.INKERHARDWARETYPE] OF
(* 		GVL.SWPWTR_TIME:
			//GVL.mb_Output_Registers[GVL.REALTIME_PLC_A2D] :=	0;	//nothing to read with FB circuit, just move motor
			IF GVL.mb_Output_Coils[GVL.REALTIME_ADVANCE] THEN		//move the motor forward
				IF TRUE THEN							//test the FB for limit - can't do this, pass through
					GVL.mb_Output_Coils[GVL.InkSweepRUN +(FTN7 * GVL.BOOLRUNTIMEGROUPSIZE)] := 	TRUE; //next RUN will force to console target
					GVL_IO.InkMotorFwd[FTN7] := TRUE;				// turn on the advance output
					GVL_IO.InkMotorRvs[FTN7] := FALSE;
					wCycleCount := wCycleCount + 1;
					IF wCycleCount > wMotorTimeOn THEN				//done with timer?
						GVL_IO.InkMotorFwd[FTN7] := FALSE;		//turn off outputs
						GVL_IO.InkMotorRvs[FTN7] := FALSE;
						GVL.mb_Output_Coils[GVL.REALTIME_ADVANCE] := FALSE; // reset the advance boolean
						wCycleCount := 0;					//reset the timer counter						
					END_IF
				END_IF
			END_IF
			IF GVL.mb_Output_Coils[GVL.REALTIME_RETARD] THEN
				IF TRUE THEN							//test the FB for limit - can't do this, pass through
					GVL.mb_Output_Coils[GVL.InkSweepRUN +(FTN7 * GVL.BOOLRUNTIMEGROUPSIZE)] := 	TRUE; //next RUN will force to console target
					GVL_IO.InkMotorFwd[FTN7] := FALSE;				// turn on the reverse output
					GVL_IO.InkMotorRvs[FTN7] := TRUE;
					wCycleCount := wCycleCount + 1;
					IF wCycleCount > wMotorTimeOn THEN				//done with timer?
						GVL_IO.InkMotorFwd[FTN7] := FALSE;		//turn off outputs
						GVL_IO.InkMotorRvs[FTN7] := FALSE;
						GVL.mb_Output_Coils[GVL.REALTIME_RETARD] := FALSE; // reset the reverse boolean
						wCycleCount := 0;					//reset the timer counter						
					END_IF
				END_IF
			END_IF
		GVL.SWPWTR_FB:
			GVL.mb_Output_Registers[GVL.REALTIME_PLC_A2D] :=	INT_TO_WORD(GVL_IO.InkInput[FTN7]);
			IF GVL.mb_Output_Coils[GVL.REALTIME_ADVANCE] THEN		//move the motor forward
				IF INT_TO_WORD(GVL_IO.InkInput[FTN7]) < 32000 THEN				//test the FB for limit - assumes 32767 is max of 10 VDC
					GVL.mb_Output_Coils[GVL.InkSweepRUN +(FTN7 * GVL.BOOLRUNTIMEGROUPSIZE)] := 	TRUE; //next RUN will force to console target
					GVL_IO.InkMotorFwd[FTN7] := TRUE;				// turn on the advance output
					GVL_IO.InkMotorRvs[FTN7] := FALSE;
					wCycleCount := wCycleCount + 1;
					IF wCycleCount > wMotorTimeOn THEN				//done with timer?
						GVL_IO.InkMotorFwd[FTN7] := FALSE;		//turn off outputs
						GVL_IO.InkMotorRvs[FTN7] := FALSE;
						GVL.mb_Output_Coils[GVL.REALTIME_ADVANCE] := FALSE; // reset the advance boolean
						wCycleCount := 0;					//reset the timer counter	
						//  curr % sweep   curr ticks - min tick allowed      max sweep %            max ticks allowed      min ticks allowed
						GVL.mb_Output_Registers[GVL.SWEEPTRIMONPRESS + (FTN7 * GVL.WORDRUNTIMEGROUPSIZE)]	:= (INT_TO_WORD(GVL_IO.InkInput[FTN7]) - GVL.w_InkInputIntMin[FTN7]) * 
								(GVL.mb_Output_Registers[GVL.MAXSWEEPTRIM]+1) / (GVL.w_InkInputIntMax[FTN7] - GVL.w_InkInputIntMin[FTN7]);
						//need the onpress setting pointed to the current % sweep of the positioner
					END_IF
				END_IF
			END_IF
			IF GVL.mb_Output_Coils[GVL.REALTIME_RETARD] THEN
				IF INT_TO_WORD(GVL_IO.InkInput[FTN7]) > 800 THEN				//test the FB for limit - assumes 32767 is max of 10 VDC
					GVL.mb_Output_Coils[GVL.InkSweepRUN +(FTN7 * GVL.BOOLRUNTIMEGROUPSIZE)] := 	TRUE; //next RUN will force to console target
					GVL_IO.InkMotorFwd[FTN7] := FALSE;				// turn on the reverse output
					GVL_IO.InkMotorRvs[FTN7] := TRUE;
					wCycleCount := wCycleCount + 1;
					IF wCycleCount > wMotorTimeOn THEN				//done with timer?
						GVL_IO.InkMotorFwd[FTN7] := FALSE;		//turn off outputs
						GVL_IO.InkMotorRvs[FTN7] := FALSE;
						GVL.mb_Output_Coils[GVL.REALTIME_RETARD] := FALSE; // reset the reverse boolean
						wCycleCount := 0;					//reset the timer counter						
						//  curr % sweep   curr ticks - min tick allowed      max sweep %            max ticks allowed      min ticks allowed
						GVL.mb_Output_Registers[GVL.SWEEPTRIMONPRESS + (FTN7 * GVL.WORDRUNTIMEGROUPSIZE)]	:= (INT_TO_WORD(GVL_IO.InkInput[FTN7]) - GVL.w_InkInputIntMin[FTN7]) * 
								(GVL.mb_Output_Registers[GVL.MAXSWEEPTRIM]+1) / (GVL.w_InkInputIntMax[FTN7] - GVL.w_InkInputIntMin[FTN7]);
						//need the onpress setting pointed to the current % sweep of the positioner
					END_IF
				END_IF
			END_IF
		GVL.SWPWTR_OUTPUT:
			GVL.mb_Output_Registers[GVL.REALTIME_PLC_A2D] :=	INT_TO_WORD(GVL_IO.InkSweepOut[FTN7]);
			IF( GVL.b_DINTInput) THEN									//how big should the adv / ret control increment be?
				w_output_incr :=  DINT_TO_INT(GVL.d_DINT10V / 100);
			ELSE
				w_output_incr := (GVL.i_INT10V / 100);
			END_IF
			IF GVL.mb_Output_Coils[GVL.REALTIME_ADVANCE] THEN
				IF GVL_IO.InkSweepOut[FTN7] < (w_output_incr *100) THEN
					GVL.mb_Output_Coils[GVL.InkSweepRUN +(FTN7 * GVL.BOOLRUNTIMEGROUPSIZE)] := 	TRUE; //next RUN will force to console target
					GVL_IO.InkSweepOut[FTN7] := GVL_IO.InkSweepOut[FTN7] + w_output_incr;
				END_IF
				GVL.mb_Output_Coils[GVL.REALTIME_ADVANCE] := FALSE;
			END_IF
			IF GVL.mb_Output_Coils[GVL.REALTIME_RETARD] THEN
				IF GVL_IO.InkSweepOut[FTN7] > w_output_incr THEN
					GVL.mb_Output_Coils[GVL.InkSweepRUN +(FTN7 * GVL.BOOLRUNTIMEGROUPSIZE)] := 	TRUE; //next RUN will force to console target
					GVL_IO.InkSweepOut[FTN7] := GVL_IO.InkSweepOut[FTN7] - w_output_incr;
				END_IF
				GVL.mb_Output_Coils[GVL.REALTIME_RETARD] := FALSE;
			END_IF			
 *)
		GVL.SWPWTR_BRIDGE:
		END_CASE
	 8:	Index := FTN8;		//assign temp index
		CASE GVL.mb_Output_Registers[GVL.INKERHARDWARETYPE] OF
(* 		GVL.SWPWTR_TIME:
			//GVL.mb_Output_Registers[GVL.REALTIME_PLC_A2D] :=	0;	//nothing to read with FB circuit, just move motor
			IF GVL.mb_Output_Coils[GVL.REALTIME_ADVANCE] THEN		//move the motor forward
				IF TRUE THEN							//test the FB for limit - can't do this, pass through
					GVL.mb_Output_Coils[GVL.InkSweepRUN +(FTN8 * GVL.BOOLRUNTIMEGROUPSIZE)] := 	TRUE; //next RUN will force to console target
					GVL_IO.InkMotorFwd[FTN8] := TRUE;				// turn on the advance output
					GVL_IO.InkMotorRvs[FTN8] := FALSE;
					wCycleCount := wCycleCount + 1;
					IF wCycleCount > wMotorTimeOn THEN				//done with timer?
						GVL_IO.InkMotorFwd[FTN8] := FALSE;		//turn off outputs
						GVL_IO.InkMotorRvs[FTN8] := FALSE;
						GVL.mb_Output_Coils[GVL.REALTIME_ADVANCE] := FALSE; // reset the advance boolean
						wCycleCount := 0;					//reset the timer counter						
					END_IF
				END_IF
			END_IF
			IF GVL.mb_Output_Coils[GVL.REALTIME_RETARD] THEN
				IF TRUE THEN							//test the FB for limit - can't do this, pass through
					GVL.mb_Output_Coils[GVL.InkSweepRUN +(FTN8 * GVL.BOOLRUNTIMEGROUPSIZE)] := 	TRUE; //next RUN will force to console target
					GVL_IO.InkMotorFwd[FTN8] := FALSE;				// turn on the reverse output
					GVL_IO.InkMotorRvs[FTN8] := TRUE;
					wCycleCount := wCycleCount + 1;
					IF wCycleCount > wMotorTimeOn THEN				//done with timer?
						GVL_IO.InkMotorFwd[FTN8] := FALSE;		//turn off outputs
						GVL_IO.InkMotorRvs[FTN8] := FALSE;
						GVL.mb_Output_Coils[GVL.REALTIME_RETARD] := FALSE; // reset the reverse boolean
						wCycleCount := 0;					//reset the timer counter						
					END_IF
				END_IF
			END_IF
		GVL.SWPWTR_FB:
			GVL.mb_Output_Registers[GVL.REALTIME_PLC_A2D] :=	INT_TO_WORD(GVL_IO.InkInput[FTN8]);
			IF GVL.mb_Output_Coils[GVL.REALTIME_ADVANCE] THEN		//move the motor forward
				IF INT_TO_WORD(GVL_IO.InkInput[FTN8]) < 32000 THEN				//test the FB for limit - assumes 32767 is max of 10 VDC
					GVL.mb_Output_Coils[GVL.InkSweepRUN +(FTN8 * GVL.BOOLRUNTIMEGROUPSIZE)] := 	TRUE; //next RUN will force to console target
					GVL_IO.InkMotorFwd[FTN8] := TRUE;				// turn on the advance output
					GVL_IO.InkMotorRvs[FTN8] := FALSE;
					wCycleCount := wCycleCount + 1;
					IF wCycleCount > wMotorTimeOn THEN				//done with timer?
						GVL_IO.InkMotorFwd[FTN8] := FALSE;		//turn off outputs
						GVL_IO.InkMotorRvs[FTN8] := FALSE;
						GVL.mb_Output_Coils[GVL.REALTIME_ADVANCE] := FALSE; // reset the advance boolean
						wCycleCount := 0;					//reset the timer counter	
						//  curr % sweep   curr ticks - min tick allowed      max sweep %            max ticks allowed      min ticks allowed
						GVL.mb_Output_Registers[GVL.SWEEPTRIMONPRESS + (FTN8 * GVL.WORDRUNTIMEGROUPSIZE)]	:= (INT_TO_WORD(GVL_IO.InkInput[FTN8]) - GVL.w_InkInputIntMin[FTN8]) * 
								(GVL.mb_Output_Registers[GVL.MAXSWEEPTRIM]+1) / (GVL.w_InkInputIntMax[FTN8] - GVL.w_InkInputIntMin[FTN8]);
						//need the onpress setting pointed to the current % sweep of the positioner
					END_IF
				END_IF
			END_IF
			IF GVL.mb_Output_Coils[GVL.REALTIME_RETARD] THEN
				IF INT_TO_WORD(GVL_IO.InkInput[FTN8]) > 800 THEN				//test the FB for limit - assumes 32767 is max of 10 VDC
					GVL.mb_Output_Coils[GVL.InkSweepRUN +(FTN8 * GVL.BOOLRUNTIMEGROUPSIZE)] := 	TRUE; //next RUN will force to console target
					GVL_IO.InkMotorFwd[FTN8] := FALSE;				// turn on the reverse output
					GVL_IO.InkMotorRvs[FTN8] := TRUE;
					wCycleCount := wCycleCount + 1;
					IF wCycleCount > wMotorTimeOn THEN				//done with timer?
						GVL_IO.InkMotorFwd[FTN8] := FALSE;		//turn off outputs
						GVL_IO.InkMotorRvs[FTN8] := FALSE;
						GVL.mb_Output_Coils[GVL.REALTIME_RETARD] := FALSE; // reset the reverse boolean
						wCycleCount := 0;					//reset the timer counter						
						//  curr % sweep   curr ticks - min tick allowed      max sweep %            max ticks allowed      min ticks allowed
						GVL.mb_Output_Registers[GVL.SWEEPTRIMONPRESS + (FTN8 * GVL.WORDRUNTIMEGROUPSIZE)]	:= (INT_TO_WORD(GVL_IO.InkInput[FTN8]) - GVL.w_InkInputIntMin[FTN8]) * 
								(GVL.mb_Output_Registers[GVL.MAXSWEEPTRIM]+1) / (GVL.w_InkInputIntMax[FTN8] - GVL.w_InkInputIntMin[FTN8]);
						//need the onpress setting pointed to the current % sweep of the positioner
					END_IF
				END_IF
			END_IF
		GVL.SWPWTR_OUTPUT:
			GVL.mb_Output_Registers[GVL.REALTIME_PLC_A2D] :=	INT_TO_WORD(GVL_IO.InkSweepOut[FTN8]);
			IF( GVL.b_DINTInput) THEN									//how big should the adv / ret control increment be?
				w_output_incr :=  DINT_TO_INT(GVL.d_DINT10V / 100);
			ELSE
				w_output_incr := (GVL.i_INT10V / 100);
			END_IF
			IF GVL.mb_Output_Coils[GVL.REALTIME_ADVANCE] THEN
				IF GVL_IO.InkSweepOut[FTN8] < (w_output_incr *100) THEN
					GVL.mb_Output_Coils[GVL.InkSweepRUN +(FTN8 * GVL.BOOLRUNTIMEGROUPSIZE)] := 	TRUE; //next RUN will force to console target
					GVL_IO.InkSweepOut[FTN8] := GVL_IO.InkSweepOut[FTN8] + w_output_incr;
				END_IF
				GVL.mb_Output_Coils[GVL.REALTIME_ADVANCE] := FALSE;
			END_IF
			IF GVL.mb_Output_Coils[GVL.REALTIME_RETARD] THEN
				IF GVL_IO.InkSweepOut[FTN8] > w_output_incr THEN
					GVL.mb_Output_Coils[GVL.InkSweepRUN +(FTN8 * GVL.BOOLRUNTIMEGROUPSIZE)] := 	TRUE; //next RUN will force to console target
					GVL_IO.InkSweepOut[FTN8] := GVL_IO.InkSweepOut[FTN8] - w_output_incr;
				END_IF
				GVL.mb_Output_Coils[GVL.REALTIME_RETARD] := FALSE;
			END_IF			
 *)
		GVL.SWPWTR_BRIDGE:
		END_CASE
	 9:	Index := FTN9;		//assign temp index
		CASE GVL.mb_Output_Registers[GVL.INKERHARDWARETYPE] OF
(* 		GVL.SWPWTR_TIME:
			//GVL.mb_Output_Registers[GVL.REALTIME_PLC_A2D] :=	0;	//nothing to read with FB circuit, just move motor
			IF GVL.mb_Output_Coils[GVL.REALTIME_ADVANCE] THEN		//move the motor forward
				IF TRUE THEN							//test the FB for limit - can't do this, pass through
					GVL.mb_Output_Coils[GVL.InkSweepRUN +(FTN9 * GVL.BOOLRUNTIMEGROUPSIZE)] := 	TRUE; //next RUN will force to console target
					GVL_IO.InkMotorFwd[FTN9] := TRUE;				// turn on the advance output
					GVL_IO.InkMotorRvs[FTN9] := FALSE;
					wCycleCount := wCycleCount + 1;
					IF wCycleCount > wMotorTimeOn THEN				//done with timer?
						GVL_IO.InkMotorFwd[FTN9] := FALSE;		//turn off outputs
						GVL_IO.InkMotorRvs[FTN9] := FALSE;
						GVL.mb_Output_Coils[GVL.REALTIME_ADVANCE] := FALSE; // reset the advance boolean
						wCycleCount := 0;					//reset the timer counter						
					END_IF
				END_IF
			END_IF
			IF GVL.mb_Output_Coils[GVL.REALTIME_RETARD] THEN
				IF TRUE THEN							//test the FB for limit - can't do this, pass through
					GVL.mb_Output_Coils[GVL.InkSweepRUN +(FTN9 * GVL.BOOLRUNTIMEGROUPSIZE)] := 	TRUE; //next RUN will force to console target
					GVL_IO.InkMotorFwd[FTN9] := FALSE;				// turn on the reverse output
					GVL_IO.InkMotorRvs[FTN9] := TRUE;
					wCycleCount := wCycleCount + 1;
					IF wCycleCount > wMotorTimeOn THEN				//done with timer?
						GVL_IO.InkMotorFwd[FTN9] := FALSE;		//turn off outputs
						GVL_IO.InkMotorRvs[FTN9] := FALSE;
						GVL.mb_Output_Coils[GVL.REALTIME_RETARD] := FALSE; // reset the reverse boolean
						wCycleCount := 0;					//reset the timer counter						
					END_IF
				END_IF
			END_IF
		GVL.SWPWTR_FB:
			GVL.mb_Output_Registers[GVL.REALTIME_PLC_A2D] :=	INT_TO_WORD(GVL_IO.InkInput[FTN9]);
			IF GVL.mb_Output_Coils[GVL.REALTIME_ADVANCE] THEN		//move the motor forward
				IF INT_TO_WORD(GVL_IO.InkInput[FTN9]) < 32000 THEN				//test the FB for limit - assumes 32767 is max of 10 VDC
					GVL.mb_Output_Coils[GVL.InkSweepRUN +(FTN9 * GVL.BOOLRUNTIMEGROUPSIZE)] := 	TRUE; //next RUN will force to console target
					GVL_IO.InkMotorFwd[FTN9] := TRUE;				// turn on the advance output
					GVL_IO.InkMotorRvs[FTN9] := FALSE;
					wCycleCount := wCycleCount + 1;
					IF wCycleCount > wMotorTimeOn THEN				//done with timer?
						GVL_IO.InkMotorFwd[FTN9] := FALSE;		//turn off outputs
						GVL_IO.InkMotorRvs[FTN9] := FALSE;
						GVL.mb_Output_Coils[GVL.REALTIME_ADVANCE] := FALSE; // reset the advance boolean
						wCycleCount := 0;					//reset the timer counter	
						//  curr % sweep   curr ticks - min tick allowed      max sweep %            max ticks allowed      min ticks allowed
						GVL.mb_Output_Registers[GVL.SWEEPTRIMONPRESS + (FTN9 * GVL.WORDRUNTIMEGROUPSIZE)]	:= (INT_TO_WORD(GVL_IO.InkInput[FTN9]) - GVL.w_InkInputIntMin[FTN9]) * 
								(GVL.mb_Output_Registers[GVL.MAXSWEEPTRIM]+1) / (GVL.w_InkInputIntMax[FTN9] - GVL.w_InkInputIntMin[FTN9]);
						//need the onpress setting pointed to the current % sweep of the positioner
					END_IF
				END_IF
			END_IF
			IF GVL.mb_Output_Coils[GVL.REALTIME_RETARD] THEN
				IF INT_TO_WORD(GVL_IO.InkInput[FTN9]) > 800 THEN				//test the FB for limit - assumes 32767 is max of 10 VDC
					GVL.mb_Output_Coils[GVL.InkSweepRUN +(FTN9 * GVL.BOOLRUNTIMEGROUPSIZE)] := 	TRUE; //next RUN will force to console target
					GVL_IO.InkMotorFwd[FTN9] := FALSE;				// turn on the reverse output
					GVL_IO.InkMotorRvs[FTN9] := TRUE;
					wCycleCount := wCycleCount + 1;
					IF wCycleCount > wMotorTimeOn THEN				//done with timer?
						GVL_IO.InkMotorFwd[FTN9] := FALSE;		//turn off outputs
						GVL_IO.InkMotorRvs[FTN9] := FALSE;
						GVL.mb_Output_Coils[GVL.REALTIME_RETARD] := FALSE; // reset the reverse boolean
						wCycleCount := 0;					//reset the timer counter						
						//  curr % sweep   curr ticks - min tick allowed      max sweep %            max ticks allowed      min ticks allowed
						GVL.mb_Output_Registers[GVL.SWEEPTRIMONPRESS + (FTN9 * GVL.WORDRUNTIMEGROUPSIZE)]	:= (INT_TO_WORD(GVL_IO.InkInput[FTN9]) - GVL.w_InkInputIntMin[FTN9]) * 
								(GVL.mb_Output_Registers[GVL.MAXSWEEPTRIM]+1) / (GVL.w_InkInputIntMax[FTN9] - GVL.w_InkInputIntMin[FTN9]);
						//need the onpress setting pointed to the current % sweep of the positioner
					END_IF
				END_IF
			END_IF
		GVL.SWPWTR_OUTPUT:
			GVL.mb_Output_Registers[GVL.REALTIME_PLC_A2D] :=	INT_TO_WORD(GVL_IO.InkSweepOut[FTN9]);
			IF( GVL.b_DINTInput) THEN									//how big should the adv / ret control increment be?
				w_output_incr :=  DINT_TO_INT(GVL.d_DINT10V / 100);
			ELSE
				w_output_incr := (GVL.i_INT10V / 100);
			END_IF
			IF GVL.mb_Output_Coils[GVL.REALTIME_ADVANCE] THEN
				IF GVL_IO.InkSweepOut[FTN9] < (w_output_incr *100) THEN
					GVL.mb_Output_Coils[GVL.InkSweepRUN +(FTN9 * GVL.BOOLRUNTIMEGROUPSIZE)] := 	TRUE; //next RUN will force to console target
					GVL_IO.InkSweepOut[FTN9] := GVL_IO.InkSweepOut[FTN9] + w_output_incr;
				END_IF
				GVL.mb_Output_Coils[GVL.REALTIME_ADVANCE] := FALSE;
			END_IF
			IF GVL.mb_Output_Coils[GVL.REALTIME_RETARD] THEN
				IF GVL_IO.InkSweepOut[FTN9] > w_output_incr THEN
					GVL.mb_Output_Coils[GVL.InkSweepRUN +(FTN9 * GVL.BOOLRUNTIMEGROUPSIZE)] := 	TRUE; //next RUN will force to console target
					GVL_IO.InkSweepOut[FTN9] := GVL_IO.InkSweepOut[FTN9] - w_output_incr;
				END_IF
				GVL.mb_Output_Coils[GVL.REALTIME_RETARD] := FALSE;
			END_IF			
 *)
		GVL.SWPWTR_BRIDGE:
		END_CASE
	 10:Index := FTN10;		//assign temp index
		CASE GVL.mb_Output_Registers[GVL.INKERHARDWARETYPE] OF
(* 		GVL.SWPWTR_TIME:
			//GVL.mb_Output_Registers[GVL.REALTIME_PLC_A2D] :=	0;	//nothing to read with FB circuit, just move motor
			IF GVL.mb_Output_Coils[GVL.REALTIME_ADVANCE] THEN		//move the motor forward
				IF TRUE THEN							//test the FB for limit - can't do this, pass through
					GVL.mb_Output_Coils[GVL.InkSweepRUN +(FTN10 * GVL.BOOLRUNTIMEGROUPSIZE)] := 	TRUE; //next RUN will force to console target
					GVL_IO.InkMotorFwd[FTN10] := TRUE;				// turn on the advance output
					GVL_IO.InkMotorRvs[FTN10] := FALSE;
					wCycleCount := wCycleCount + 1;
					IF wCycleCount > wMotorTimeOn THEN				//done with timer?
						GVL_IO.InkMotorFwd[FTN10] := FALSE;		//turn off outputs
						GVL_IO.InkMotorRvs[FTN10] := FALSE;
						GVL.mb_Output_Coils[GVL.REALTIME_ADVANCE] := FALSE; // reset the advance boolean
						wCycleCount := 0;					//reset the timer counter						
					END_IF
				END_IF
			END_IF
			IF GVL.mb_Output_Coils[GVL.REALTIME_RETARD] THEN
				IF TRUE THEN							//test the FB for limit - can't do this, pass through
					GVL.mb_Output_Coils[GVL.InkSweepRUN +(FTN10 * GVL.BOOLRUNTIMEGROUPSIZE)] := 	TRUE; //next RUN will force to console target
					GVL_IO.InkMotorFwd[FTN10] := FALSE;				// turn on the reverse output
					GVL_IO.InkMotorRvs[FTN10] := TRUE;
					wCycleCount := wCycleCount + 1;
					IF wCycleCount > wMotorTimeOn THEN				//done with timer?
						GVL_IO.InkMotorFwd[FTN10] := FALSE;		//turn off outputs
						GVL_IO.InkMotorRvs[FTN10] := FALSE;
						GVL.mb_Output_Coils[GVL.REALTIME_RETARD] := FALSE; // reset the reverse boolean
						wCycleCount := 0;					//reset the timer counter						
					END_IF
				END_IF
			END_IF
		GVL.SWPWTR_FB:
			GVL.mb_Output_Registers[GVL.REALTIME_PLC_A2D] :=	INT_TO_WORD(GVL_IO.InkInput[FTN10]);
			IF GVL.mb_Output_Coils[GVL.REALTIME_ADVANCE] THEN		//move the motor forward
				IF INT_TO_WORD(GVL_IO.InkInput[FTN10]) < 32000 THEN				//test the FB for limit - assumes 32767 is max of 10 VDC
					GVL.mb_Output_Coils[GVL.InkSweepRUN +(FTN10 * GVL.BOOLRUNTIMEGROUPSIZE)] := 	TRUE; //next RUN will force to console target
					GVL_IO.InkMotorFwd[FTN10] := TRUE;				// turn on the advance output
					GVL_IO.InkMotorRvs[FTN10] := FALSE;
					wCycleCount := wCycleCount + 1;
					IF wCycleCount > wMotorTimeOn THEN				//done with timer?
						GVL_IO.InkMotorFwd[FTN10] := FALSE;		//turn off outputs
						GVL_IO.InkMotorRvs[FTN10] := FALSE;
						GVL.mb_Output_Coils[GVL.REALTIME_ADVANCE] := FALSE; // reset the advance boolean
						wCycleCount := 0;					//reset the timer counter	
						//  curr % sweep   curr ticks - min tick allowed      max sweep %            max ticks allowed      min ticks allowed
						GVL.mb_Output_Registers[GVL.SWEEPTRIMONPRESS + (FTN10 * GVL.WORDRUNTIMEGROUPSIZE)]	:= (INT_TO_WORD(GVL_IO.InkInput[FTN10]) - GVL.w_InkInputIntMin[FTN10]) * 
								(GVL.mb_Output_Registers[GVL.MAXSWEEPTRIM]+1) / (GVL.w_InkInputIntMax[FTN10] - GVL.w_InkInputIntMin[FTN10]);
						//need the onpress setting pointed to the current % sweep of the positioner
					END_IF
				END_IF
			END_IF
			IF GVL.mb_Output_Coils[GVL.REALTIME_RETARD] THEN
				IF INT_TO_WORD(GVL_IO.InkInput[FTN10]) > 800 THEN				//test the FB for limit - assumes 32767 is max of 10 VDC
					GVL.mb_Output_Coils[GVL.InkSweepRUN +(FTN10 * GVL.BOOLRUNTIMEGROUPSIZE)] := 	TRUE; //next RUN will force to console target
					GVL_IO.InkMotorFwd[FTN10] := FALSE;				// turn on the reverse output
					GVL_IO.InkMotorRvs[FTN10] := TRUE;
					wCycleCount := wCycleCount + 1;
					IF wCycleCount > wMotorTimeOn THEN				//done with timer?
						GVL_IO.InkMotorFwd[FTN10] := FALSE;		//turn off outputs
						GVL_IO.InkMotorRvs[FTN10] := FALSE;
						GVL.mb_Output_Coils[GVL.REALTIME_RETARD] := FALSE; // reset the reverse boolean
						wCycleCount := 0;					//reset the timer counter						
						//  curr % sweep   curr ticks - min tick allowed      max sweep %            max ticks allowed      min ticks allowed
						GVL.mb_Output_Registers[GVL.SWEEPTRIMONPRESS + (FTN10 * GVL.WORDRUNTIMEGROUPSIZE)]	:= (INT_TO_WORD(GVL_IO.InkInput[FTN10]) - GVL.w_InkInputIntMin[FTN10]) * 
								(GVL.mb_Output_Registers[GVL.MAXSWEEPTRIM]+1) / (GVL.w_InkInputIntMax[FTN10] - GVL.w_InkInputIntMin[FTN10]);
						//need the onpress setting pointed to the current % sweep of the positioner
					END_IF
				END_IF
			END_IF
		GVL.SWPWTR_OUTPUT:
			GVL.mb_Output_Registers[GVL.REALTIME_PLC_A2D] :=	INT_TO_WORD(GVL_IO.InkSweepOut[FTN10]);
			IF( GVL.b_DINTInput) THEN									//how big should the adv / ret control increment be?
				w_output_incr :=  DINT_TO_INT(GVL.d_DINT10V / 100);
			ELSE
				w_output_incr := (GVL.i_INT10V / 100);
			END_IF
			IF GVL.mb_Output_Coils[GVL.REALTIME_ADVANCE] THEN
				IF GVL_IO.InkSweepOut[FTN10] < (w_output_incr *100) THEN
					GVL.mb_Output_Coils[GVL.InkSweepRUN +(FTN10 * GVL.BOOLRUNTIMEGROUPSIZE)] := 	TRUE; //next RUN will force to console target
					GVL_IO.InkSweepOut[FTN10] := GVL_IO.InkSweepOut[FTN10] + w_output_incr;
				END_IF
				GVL.mb_Output_Coils[GVL.REALTIME_ADVANCE] := FALSE;
			END_IF
			IF GVL.mb_Output_Coils[GVL.REALTIME_RETARD] THEN
				IF GVL_IO.InkSweepOut[FTN10] > w_output_incr THEN
					GVL.mb_Output_Coils[GVL.InkSweepRUN +(FTN10 * GVL.BOOLRUNTIMEGROUPSIZE)] := 	TRUE; //next RUN will force to console target
					GVL_IO.InkSweepOut[FTN10] := GVL_IO.InkSweepOut[FTN10] - w_output_incr;
				END_IF
				GVL.mb_Output_Coils[GVL.REALTIME_RETARD] := FALSE;
			END_IF			
 *)
		GVL.SWPWTR_BRIDGE:
		END_CASE

	// Water analog inputs and outputs

